// Mitsubishi GX Works2 project: BookEX6_22 Compare   PLC: Q13UDV

// global labels: Global
VAR_GLOBAL
  bVar0 AT M5000 : BOOL;
  abArray0 AT M5010 : ARRAY [0..49] OF BOOL;
  sStr0 AT D5000 : STRING[199];
  sStr1 AT D5100 : STRING[199];
  sStr2 AT D5200 : STRING[199];
  sStr3 AT D5300 : STRING[199];
  sStr4 AT D5400 : STRING[199];
  sStr5 AT D5500 : STRING[199];
  sStr6 AT D5600 : STRING[199];
  sStr7 AT D5700 : STRING[199];
  sStr8 AT D5800 : STRING[199];
  sStr9 AT D5900 : STRING[199];
  iVar0 AT D4500 : INT;
  iVar1 AT D4501 : INT;
  iVar2 AT D4502 : INT;
  iVar3 AT D4503 : INT;
  iVar4 AT D4504 : INT;
  iVar5 AT D4505 : INT;
  iVar6 AT D4506 : INT;
  iVar7 AT D4507 : INT;
  iVar8 AT D4508 : INT;
  iVar9 AT D4509 : INT;
  dVar0 AT D4510 : DINT;
  dVar1 AT D4512 : DINT;
  dVar2 AT D4514 : DINT;
  dVar3 AT D4516 : DINT;
  dVar4 AT D4518 : DINT;
  dVar5 AT D4520 : DINT;
  dVar6 AT D4522 : DINT;
  dVar7 AT D4524 : DINT;
  dVar8 AT D4526 : DINT;
  dVar9 AT D4528 : DINT;
  wVar0 AT D4530 : WORD;
  wVar1 AT D4531 : WORD;
  wVar2 AT D4532 : WORD;
  wVar3 AT D4533 : WORD;
  wVar4 AT D4534 : WORD;
  wVar5 AT D4535 : WORD;
  wVar6 AT D4536 : WORD;
  wVar7 AT D4537 : WORD;
  wVar8 AT D4538 : WORD;
  wVar9 AT D4539 : WORD;
  dwVar0 AT D4540 : DWORD;
  dwVar1 AT D4542 : DWORD;
  dwVar2 AT D4544 : DWORD;
  dwVar3 AT D4546 : DWORD;
  dwVar4 AT D4548 : DWORD;
  dwVar5 AT D4550 : DWORD;
  dwVar6 AT D4552 : DWORD;
  dwVar7 AT D4554 : DWORD;
  dwVar8 AT D4556 : DWORD;
  dwVar9 AT D4558 : DWORD;
  fsVar0 AT D4560 : REAL;
  fsVar1 AT D4562 : REAL;
  fsVar2 AT D4564 : REAL;
  fsVar3 AT D4566 : REAL;
  fsVar4 AT D4568 : REAL;
  fsVar5 AT D4570 : REAL;
  fsVar6 AT D4572 : REAL;
  fsVar7 AT D4574 : REAL;
  fsVar8 AT D4576 : REAL;
  fsVar9 AT D4578 : REAL;
  fdVar0 AT D4580 : LREAL;
  tTime0 AT D4620 : TIME;
  tTime1 AT D4622 : TIME;
  tTime2 AT D4624 : TIME;
  tTime3 AT D4626 : TIME;
  tTime4 AT D4628 : TIME;
  tTime5 AT D4630 : TIME;
  tTime6 AT D4632 : TIME;
  tTime7 AT D4634 : TIME;
  tTime8 AT D4636 : TIME;
  tTime9 AT D4638 : TIME;
  tTime10 AT D4640 : TIME;
  bVar1 AT M5001 : BOOL;
  bVar2 AT M5002 : BOOL;
  bVar3 AT M5003 : BOOL;
  bVar4 AT M5004 : BOOL;
  bVar5 AT M5005 : BOOL;
  bVar6 AT M5006 : BOOL;
  bVar7 AT M5007 : BOOL;
  bVar8 AT M5008 : BOOL;
  bVar9 AT M5009 : BOOL;
  abArray1 AT M5060 : ARRAY [0..49] OF BOOL;
  abArray2 AT M5110 : ARRAY [0..49] OF BOOL;
  abArray3 AT M5160 : ARRAY [0..49] OF BOOL;
  abArray4 AT M5210 : ARRAY [0..49] OF BOOL;
  abArray5 AT M5260 : ARRAY [0..49] OF BOOL;
  abArray6 AT M5310 : ARRAY [0..49] OF BOOL;
  abArray7 AT M5360 : ARRAY [0..49] OF BOOL;
  abArray8 AT M5410 : ARRAY [0..49] OF BOOL;
  abArray9 AT M5460 : ARRAY [0..49] OF BOOL;
  fdVar1 AT D4584 : LREAL;
  fdVar2 AT D4588 : LREAL;
  fdVar3 AT D4592 : LREAL;
  fdVar4 AT D4596 : LREAL;
  fdVar5 AT D4600 : LREAL;
  fdVar6 AT D4604 : LREAL;
  fdVar7 AT D4608 : LREAL;
  fdVar8 AT D4612 : LREAL;
  fdVar9 AT D4616 : LREAL;
  afsPen0 AT D2000 : ARRAY [0..499] OF REAL;
  afsPen1 AT D3000 : ARRAY [0..499] OF REAL;
END_VAR
// user libraries (not included): HMI

PROGRAM ExBKCMP
VAR
  Mov4WORD_1 : Mov4WORD;
  Mov4WORD_2 : Mov4WORD;
  Mov4WORD_0 : Mov4WORD;
  Mov4WORD_3 : Mov4WORD;
  Mov4WORD_4 : Mov4WORD;
END_VAR
(* structured ladder/FBD written out as ST: instructions are called as NAME(EN, inputs, outputs); _pN, _eN, _tN stand for wires *)
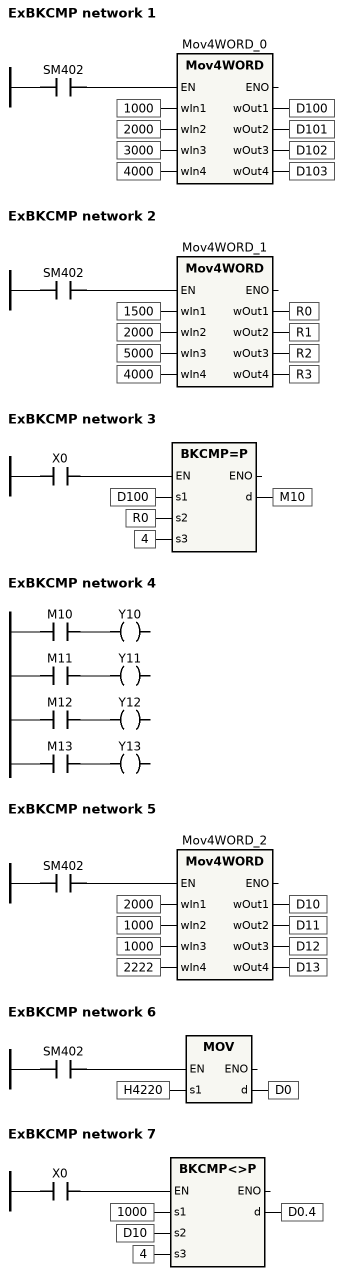
(* network 1 *)
Mov4WORD_0(EN := SM402, wIn1 := 1000, wIn2 := 2000, wIn3 := 3000, wIn4 := 4000, wOut1 => D100, wOut2 => D101, wOut3 => D102, wOut4 => D103);
(* network 2 *)
Mov4WORD_1(EN := SM402, wIn1 := 1500, wIn2 := 2000, wIn3 := 5000, wIn4 := 4000, wOut1 => R0, wOut2 => R1, wOut3 => R2, wOut4 => R3);
(* network 3 *)
BKCMP=P(X0, D100, R0, 4, M10);
(* network 4 *)
Y10 := M10;
Y11 := M11;
Y12 := M12;
Y13 := M13;
(* network 5 *)
Mov4WORD_2(EN := SM402, wIn1 := 2000, wIn2 := 1000, wIn3 := 1000, wIn4 := 2222, wOut1 => D10, wOut2 => D11, wOut3 => D12, wOut4 => D13);
(* network 6 *)
MOV(SM402, H4220, D0);
(* network 7 *)
BKCMP<>P(X0, 1000, D10, 4, D0.4);
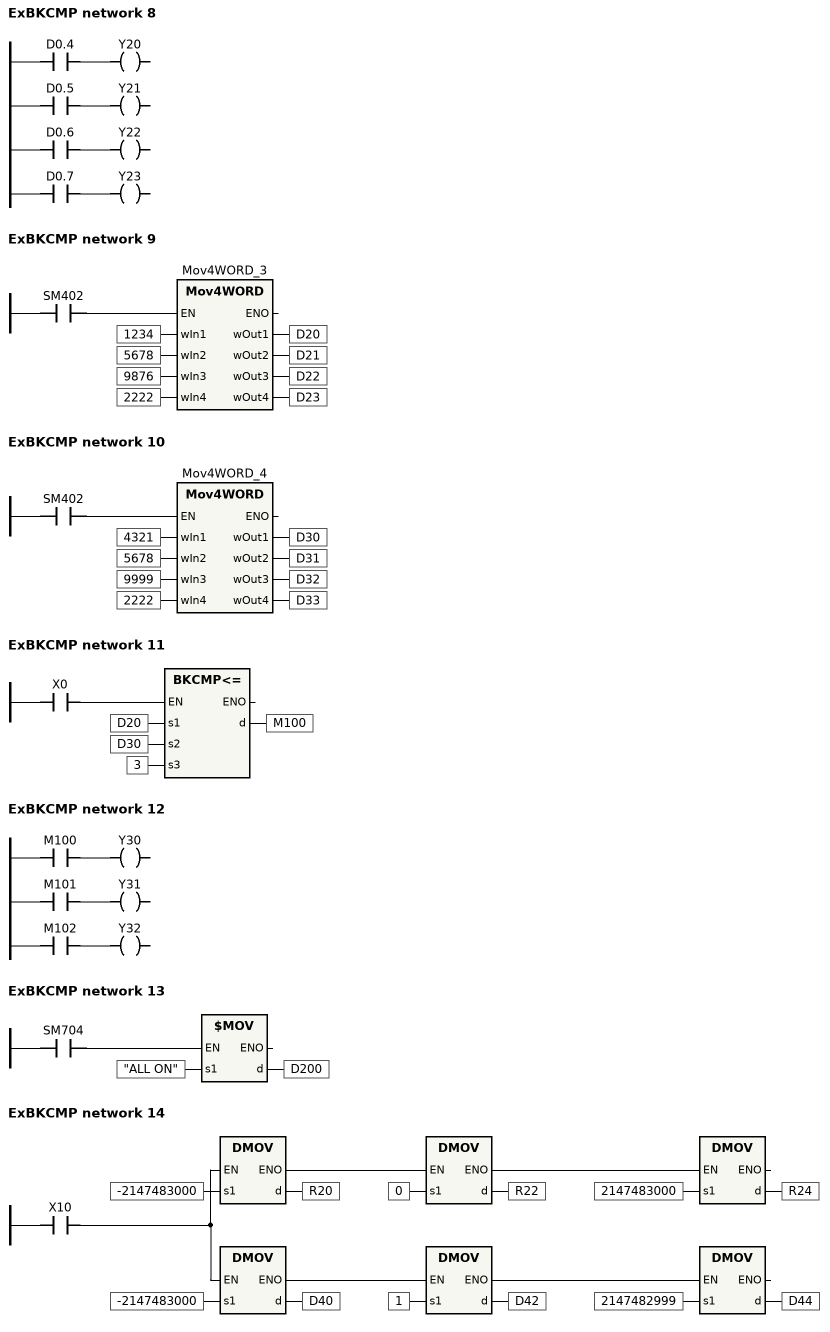
(* network 8 *)
Y20 := D0.4;
Y21 := D0.5;
Y22 := D0.6;
Y23 := D0.7;
(* network 9 *)
Mov4WORD_3(EN := SM402, wIn1 := 1234, wIn2 := 5678, wIn3 := 9876, wIn4 := 2222, wOut1 => D20, wOut2 => D21, wOut3 => D22, wOut4 => D23);
(* network 10 *)
Mov4WORD_4(EN := SM402, wIn1 := 4321, wIn2 := 5678, wIn3 := 9999, wIn4 := 2222, wOut1 => D30, wOut2 => D31, wOut3 => D32, wOut4 => D33);
(* network 11 *)
BKCMP<=(X0, D20, D30, 3, M100);
(* network 12 *)
Y30 := M100;
Y31 := M101;
Y32 := M102;
(* network 13 *)
$MOV(SM704, "ALL ON", D200);
(* network 14 *)
_e1 := DMOV(X10, -2147483000, R20);
_e2 := DMOV(_e1, 0, R22);
DMOV(_e2, 2147483000, R24);
_e3 := DMOV(X10, -2147483000, D40);
_e4 := DMOV(_e3, 1, D42);
DMOV(_e4, 2147482999, D44);
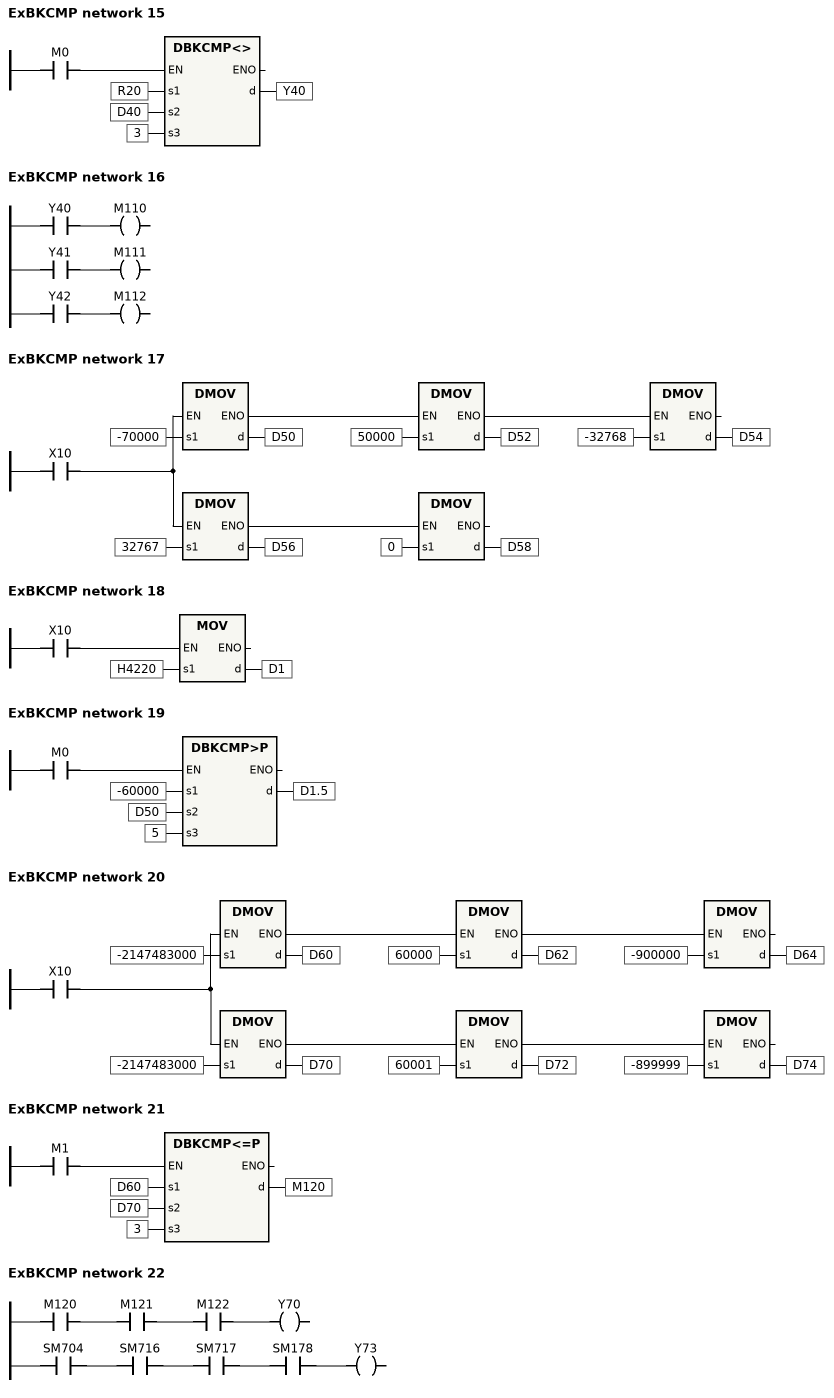
(* network 15 *)
DBKCMP<>(M0, R20, D40, 3, Y40);
(* network 16 *)
M110 := Y40;
M111 := Y41;
M112 := Y42;
(* network 17 *)
_e1 := DMOV(X10, -70000, D50);
_e2 := DMOV(_e1, 50000, D52);
DMOV(_e2, -32768, D54);
_e3 := DMOV(X10, 32767, D56);
DMOV(_e3, 0, D58);
(* network 18 *)
MOV(X10, H4220, D1);
(* network 19 *)
DBKCMP>P(M0, -60000, D50, 5, D1.5);
(* network 20 *)
_e1 := DMOV(X10, -2147483000, D60);
_e2 := DMOV(_e1, 60000, D62);
DMOV(_e2, -900000, D64);
_e3 := DMOV(X10, -2147483000, D70);
_e4 := DMOV(_e3, 60001, D72);
DMOV(_e4, -899999, D74);
(* network 21 *)
DBKCMP<=P(M1, D60, D70, 3, M120);
(* network 22 *)
Y70 := M120 AND M121 AND M122;
Y73 := SM704 AND SM716 AND SM717 AND SM178;
END_PROGRAM

PROGRAM ExCMP
VAR
  abRes : ARRAY [0..2] OF BOOL;
END_VAR
(* structured ladder/FBD written out as ST: instructions are called as NAME(EN, inputs, outputs); _pN, _eN, _tN stand for wires *)
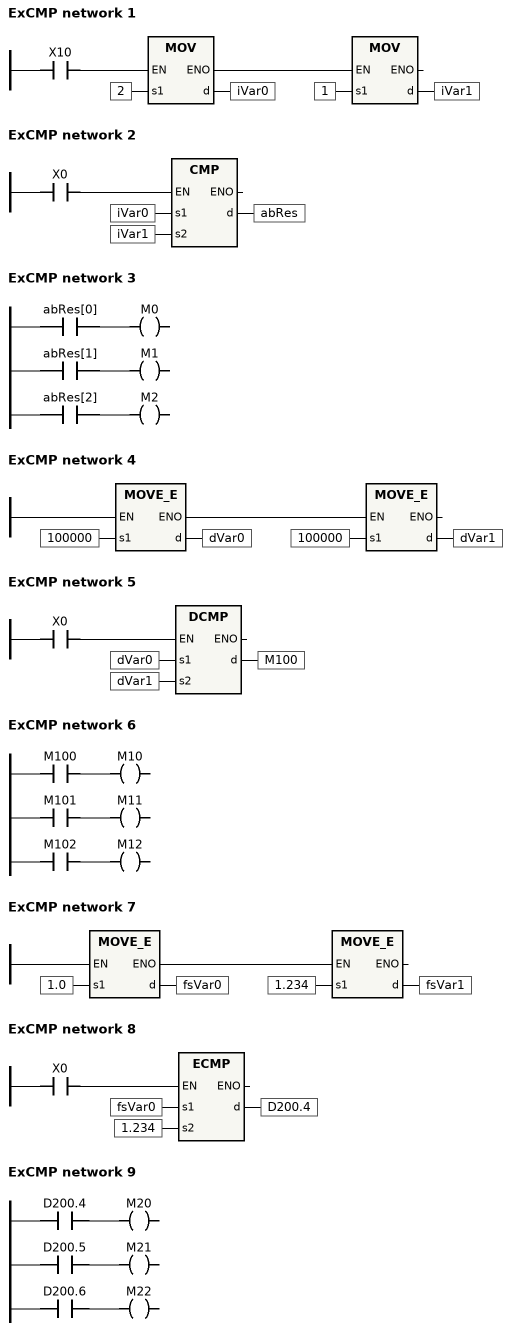
(* network 1 *)
_e1 := MOV(X10, 2, iVar0);
MOV(_e1, 1, iVar1);
(* network 2 *)
CMP(X0, iVar0, iVar1, abRes);
(* network 3 *)
M0 := abRes[0];
M1 := abRes[1];
M2 := abRes[2];
(* network 4 *)
_e1 := MOVE_E(TRUE, 100000, dVar0);
MOVE_E(_e1, 100000, dVar1);
(* network 5 *)
DCMP(X0, dVar0, dVar1, M100);
(* network 6 *)
M10 := M100;
M11 := M101;
M12 := M102;
(* network 7 *)
_e1 := MOVE_E(TRUE, 1.0, fsVar0);
MOVE_E(_e1, 1.234, fsVar1);
(* network 8 *)
ECMP(X0, fsVar0, 1.234, D200.4);
(* network 9 *)
M20 := D200.4;
M21 := D200.5;
M22 := D200.6;
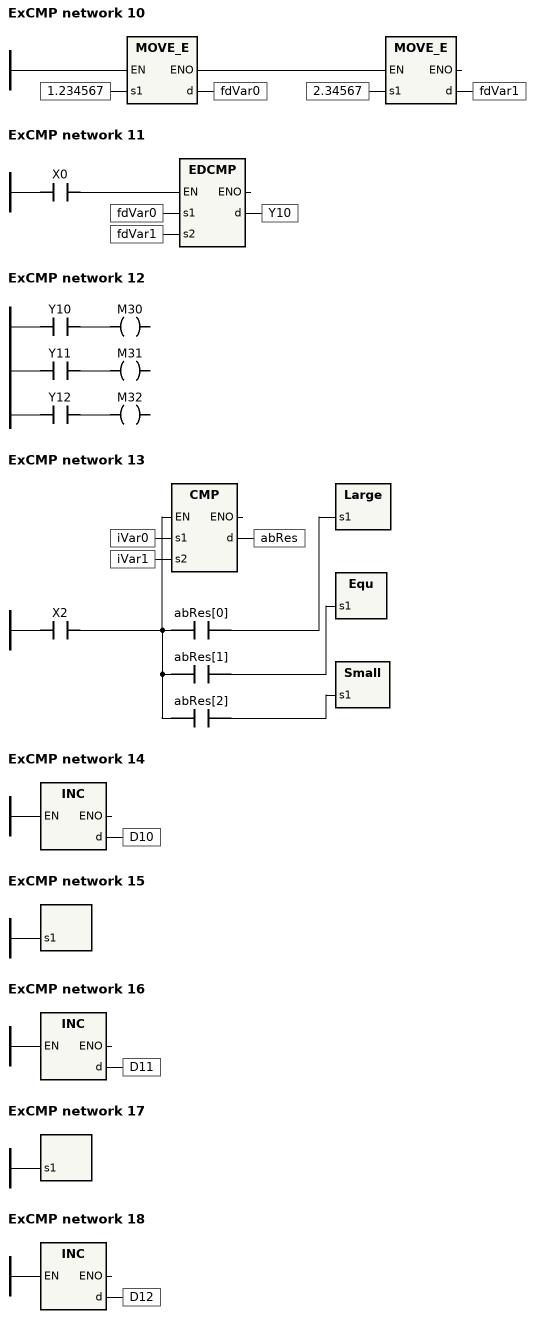
(* network 10 *)
_e1 := MOVE_E(TRUE, 1.234567, fdVar0);
MOVE_E(_e1, 2.34567, fdVar1);
(* network 11 *)
EDCMP(X0, fdVar0, fdVar1, Y10);
(* network 12 *)
M30 := Y10;
M31 := Y11;
M32 := Y12;
(* network 13 *)
CMP(X2, iVar0, iVar1, abRes);
(* element kind 9 Large <- X2 AND abRes[0] *)
(* element kind 9 Equ <- X2 AND abRes[1] *)
(* element kind 9 Small <- X2 AND abRes[2] *)
(* network 14 *)
INC(TRUE, D10);
(* network 15 *)
(* element kind 10  <- TRUE *)
(* network 16 Large: *)
INC(TRUE, D11);
(* network 17 *)
(* element kind 10  <- TRUE *)
(* network 18 Equ: *)
INC(TRUE, D12);
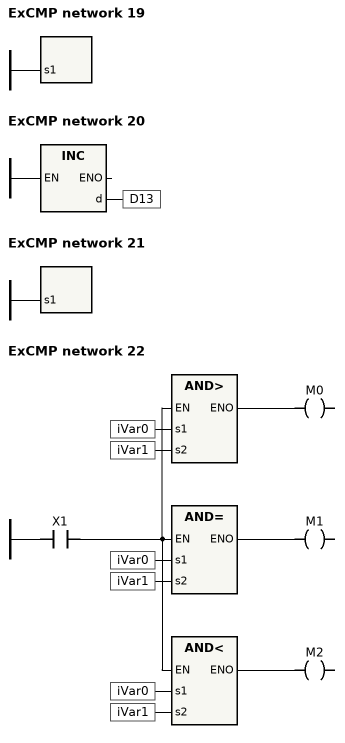
(* network 19 *)
(* element kind 10  <- TRUE *)
(* network 20 Small: *)
INC(TRUE, D13);
(* network 21 *)
(* element kind 10  <- TRUE *)
(* network 22 *)
_e1 := AND>(X1, iVar0, iVar1);
M0 := _e1;
_e2 := AND=(X1, iVar0, iVar1);
M1 := _e2;
_e3 := AND<(X1, iVar0, iVar1);
M2 := _e3;
END_PROGRAM

PROGRAM ExLD
(* structured ladder/FBD written out as ST: instructions are called as NAME(EN, inputs, outputs); _pN, _eN, _tN stand for wires *)
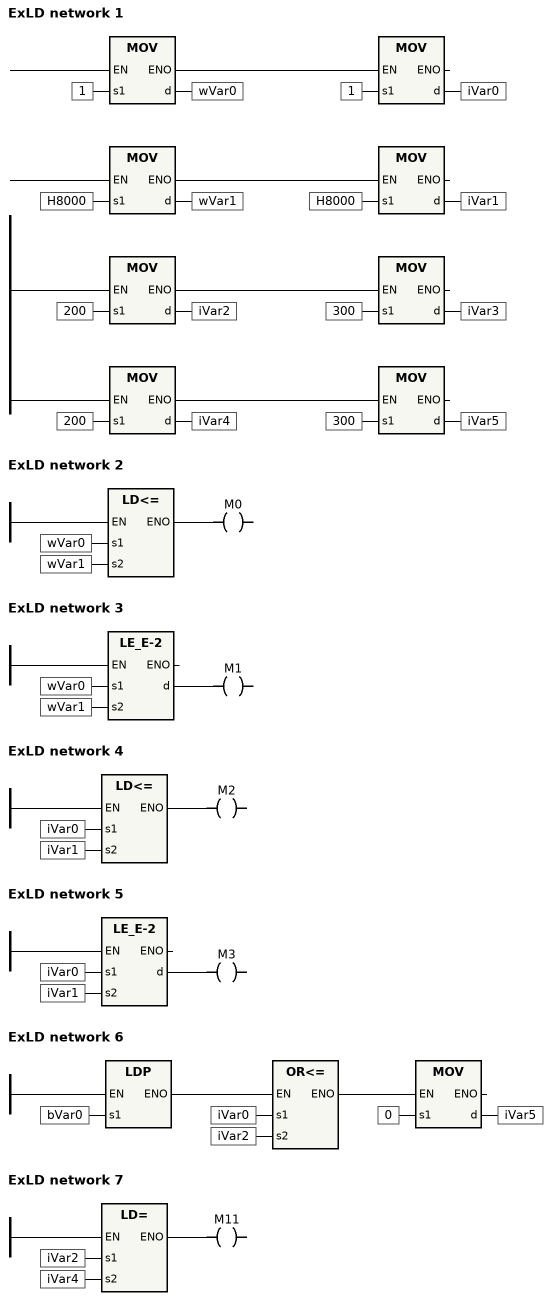
(* network 1 *)
_e1 := MOV(TRUE, 1, wVar0);
MOV(_e1, 1, iVar0);
_e2 := MOV(TRUE, H8000, wVar1);
MOV(_e2, H8000, iVar1);
_e3 := MOV(TRUE, 200, iVar2);
MOV(_e3, 300, iVar3);
_e4 := MOV(TRUE, 200, iVar4);
MOV(_e4, 300, iVar5);
(* network 2 *)
_e1 := LD<=(TRUE, wVar0, wVar1);
M0 := _e1;
(* network 3 *)
LE_E(TRUE, wVar0, wVar1, _t1);
M1 := _t1;
(* network 4 *)
_e1 := LD<=(TRUE, iVar0, iVar1);
M2 := _e1;
(* network 5 *)
LE_E(TRUE, iVar0, iVar1, _t1);
M3 := _t1;
(* network 6 *)
_e1 := LDP(TRUE, bVar0);
_e2 := OR<=(_e1, iVar0, iVar2);
MOV(_e2, 0, iVar5);
(* network 7 *)
_e1 := LD=(TRUE, iVar2, iVar4);
M11 := _e1;
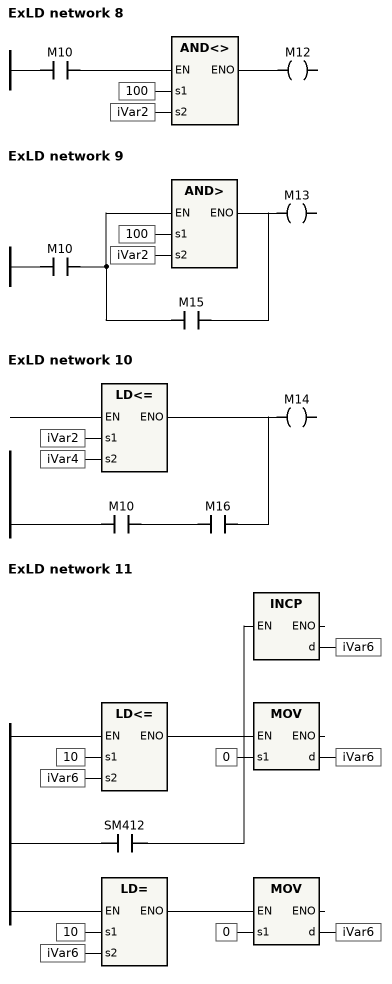
(* network 8 *)
_e1 := AND<>(M10, 100, iVar2);
M12 := _e1;
(* network 9 *)
_e1 := AND>(M10, 100, iVar2);
M13 := _e1 OR (M10 AND M15);
(* network 10 *)
_e1 := LD<=(TRUE, iVar2, iVar4);
M14 := (M10 AND M16) OR _e1;
(* network 11 *)
INCP(SM412, iVar6);
_e1 := LD<=(TRUE, 10, iVar6);
MOV(_e1, 0, iVar6);
_e2 := LD=(TRUE, 10, iVar6);
MOV(_e2, 0, iVar6);
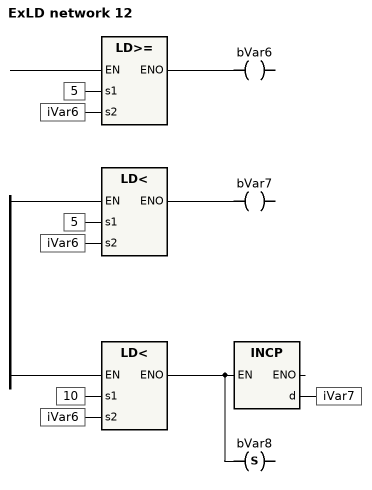
(* network 12 *)
_e1 := LD>=(TRUE, 5, iVar6);
bVar6 := _e1;
_e2 := LD<(TRUE, 5, iVar6);
bVar7 := _e2;
_e3 := LD<(TRUE, 10, iVar6);
SET(_e3, bVar8);
INCP(_e3, iVar7);
END_PROGRAM

PROGRAM ExLD$
(* structured ladder/FBD written out as ST: instructions are called as NAME(EN, inputs, outputs); _pN, _eN, _tN stand for wires *)
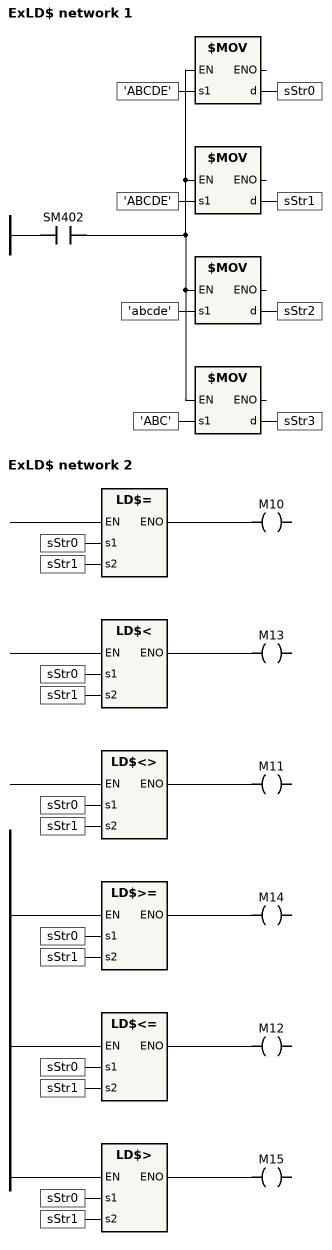
(* network 1 *)
$MOV(SM402, 'ABCDE', sStr0);
$MOV(SM402, 'ABCDE', sStr1);
$MOV(SM402, 'abcde', sStr2);
$MOV(SM402, 'ABC', sStr3);
(* network 2 *)
_e1 := LD$=(TRUE, sStr0, sStr1);
M10 := _e1;
_e2 := LD$<(TRUE, sStr0, sStr1);
M13 := _e2;
_e3 := LD$<>(TRUE, sStr0, sStr1);
M11 := _e3;
_e4 := LD$>=(TRUE, sStr0, sStr1);
M14 := _e4;
_e5 := LD$<=(TRUE, sStr0, sStr1);
M12 := _e5;
_e6 := LD$>(TRUE, sStr0, sStr1);
M15 := _e6;
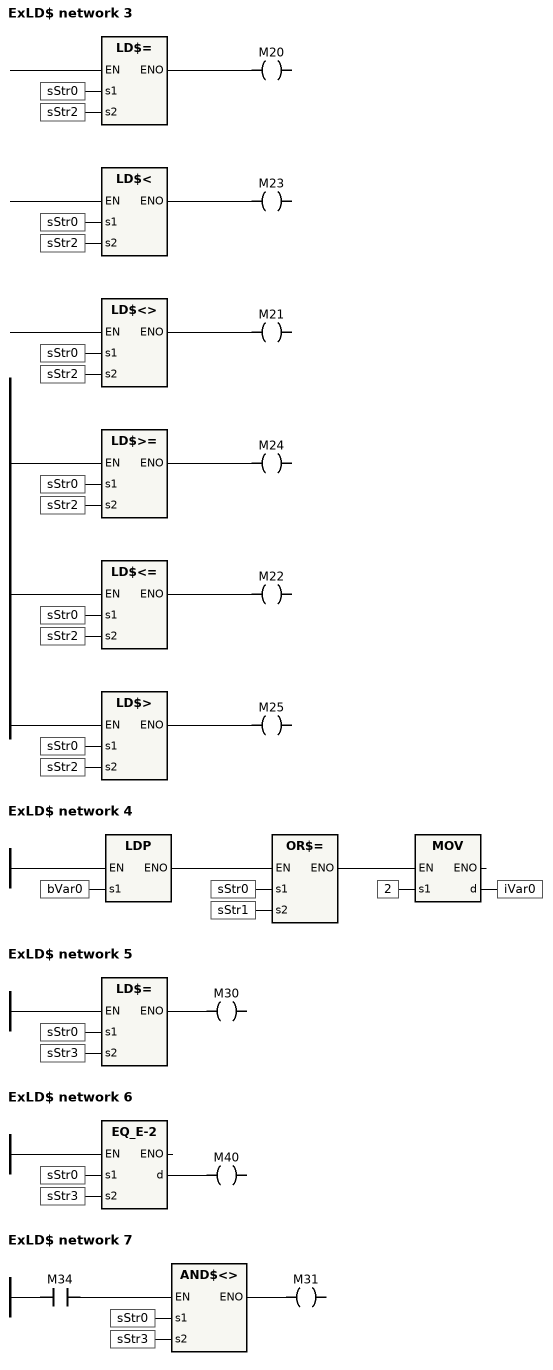
(* network 3 *)
_e1 := LD$=(TRUE, sStr0, sStr2);
M20 := _e1;
_e2 := LD$<(TRUE, sStr0, sStr2);
M23 := _e2;
_e3 := LD$<>(TRUE, sStr0, sStr2);
M21 := _e3;
_e4 := LD$>=(TRUE, sStr0, sStr2);
M24 := _e4;
_e5 := LD$<=(TRUE, sStr0, sStr2);
M22 := _e5;
_e6 := LD$>(TRUE, sStr0, sStr2);
M25 := _e6;
(* network 4 *)
_e1 := LDP(TRUE, bVar0);
_e2 := OR$=(_e1, sStr0, sStr1);
MOV(_e2, 2, iVar0);
(* network 5 *)
_e1 := LD$=(TRUE, sStr0, sStr3);
M30 := _e1;
(* network 6 *)
EQ_E(TRUE, sStr0, sStr3, _t1);
M40 := _t1;
(* network 7 *)
_e1 := AND$<>(M34, sStr0, sStr3);
M31 := _e1;
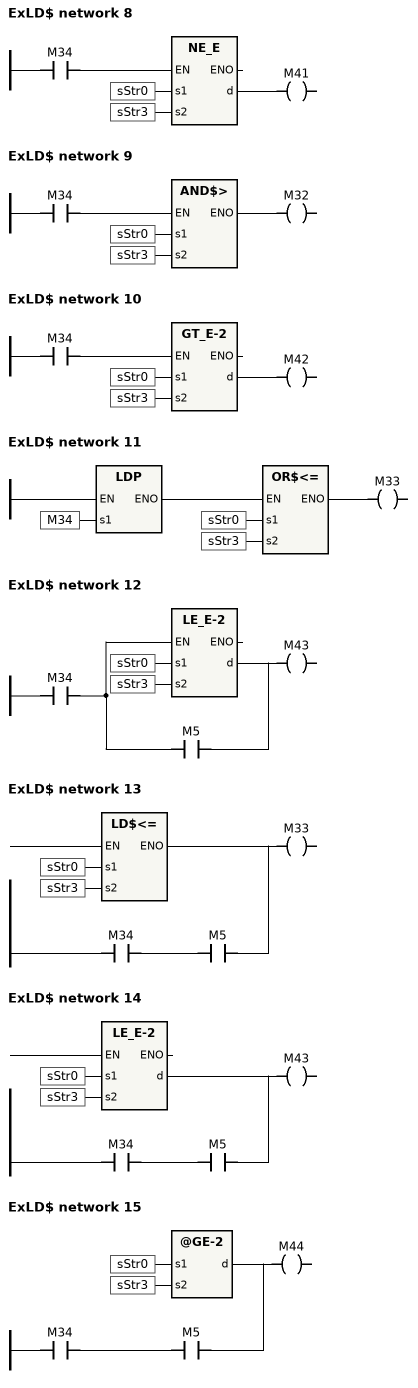
(* network 8 *)
NE_E(M34, sStr0, sStr3, _t1);
M41 := _t1;
(* network 9 *)
_e1 := AND$>(M34, sStr0, sStr3);
M32 := _e1;
(* network 10 *)
GT_E(M34, sStr0, sStr3, _t1);
M42 := _t1;
(* network 11 *)
_e1 := LDP(TRUE, M34);
_e2 := OR$<=(_e1, sStr0, sStr3);
M33 := _e2;
(* network 12 *)
LE_E(M34, sStr0, sStr3, _t1);
M43 := (M34 AND M5) OR _t1;
(* network 13 *)
_e1 := LD$<=(TRUE, sStr0, sStr3);
M33 := (M34 AND M5) OR _e1;
(* network 14 *)
LE_E(TRUE, sStr0, sStr3, _t1);
M43 := (M34 AND M5) OR _t1;
(* network 15 *)
M44 := (M34 AND M5) OR (@GE-2(sStr0, sStr3));
END_PROGRAM

PROGRAM ExLDD
(* structured ladder/FBD written out as ST: instructions are called as NAME(EN, inputs, outputs); _pN, _eN, _tN stand for wires *)
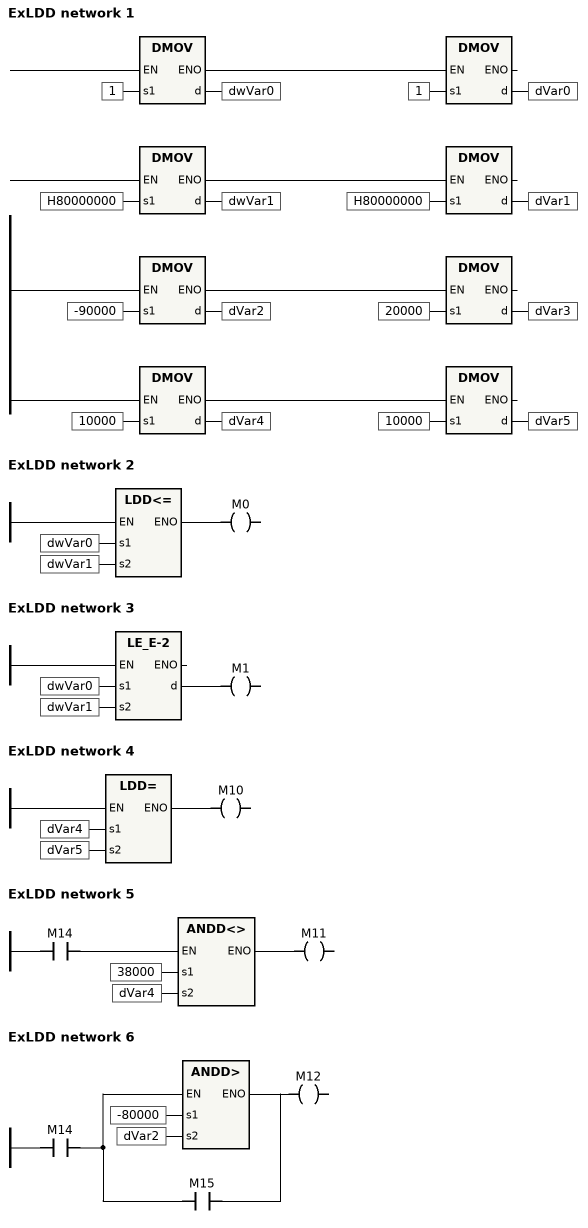
(* network 1 *)
_e1 := DMOV(TRUE, 1, dwVar0);
DMOV(_e1, 1, dVar0);
_e2 := DMOV(TRUE, H80000000, dwVar1);
DMOV(_e2, H80000000, dVar1);
_e3 := DMOV(TRUE, -90000, dVar2);
DMOV(_e3, 20000, dVar3);
_e4 := DMOV(TRUE, 10000, dVar4);
DMOV(_e4, 10000, dVar5);
(* network 2 *)
_e1 := LDD<=(TRUE, dwVar0, dwVar1);
M0 := _e1;
(* network 3 *)
LE_E(TRUE, dwVar0, dwVar1, _t1);
M1 := _t1;
(* network 4 *)
_e1 := LDD=(TRUE, dVar4, dVar5);
M10 := _e1;
(* network 5 *)
_e1 := ANDD<>(M14, 38000, dVar4);
M11 := _e1;
(* network 6 *)
_e1 := ANDD>(M14, -80000, dVar2);
M12 := _e1 OR (M14 AND M15);
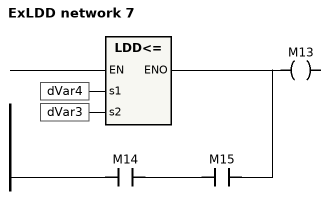
(* network 7 *)
_e1 := LDD<=(TRUE, dVar4, dVar3);
M13 := (M14 AND M15) OR _e1;
END_PROGRAM

PROGRAM ExLDE
(* structured ladder/FBD written out as ST: instructions are called as NAME(EN, inputs, outputs); _pN, _eN, _tN stand for wires *)
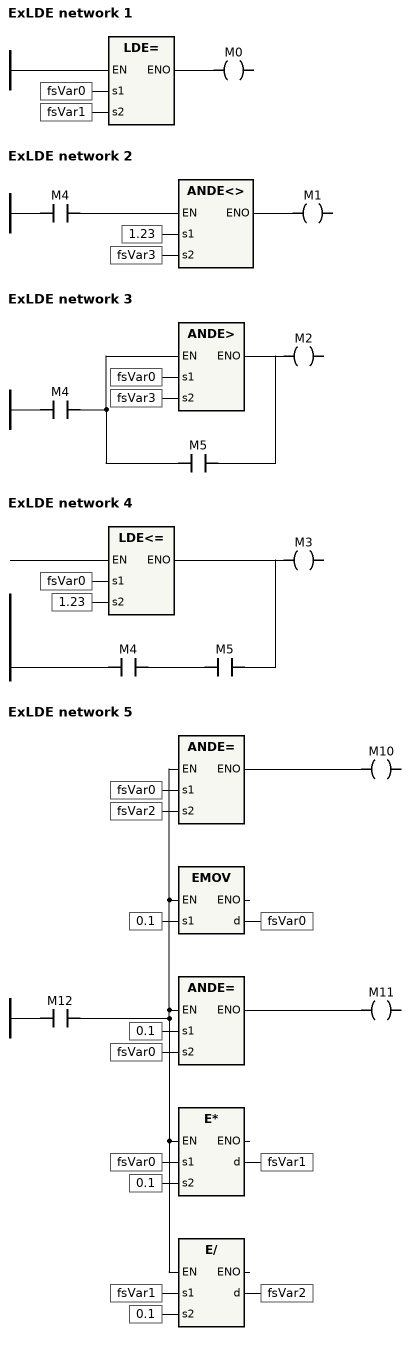
(* network 1 *)
_e1 := LDE=(TRUE, fsVar0, fsVar1);
M0 := _e1;
(* network 2 *)
_e1 := ANDE<>(M4, 1.23, fsVar3);
M1 := _e1;
(* network 3 *)
_e1 := ANDE>(M4, fsVar0, fsVar3);
M2 := _e1 OR (M4 AND M5);
(* network 4 *)
_e1 := LDE<=(TRUE, fsVar0, 1.23);
M3 := (M4 AND M5) OR _e1;
(* network 5 *)
EMOV(M12, 0.1, fsVar0);
E*(M12, fsVar0, 0.1, fsVar1);
E/(M12, fsVar1, 0.1, fsVar2);
_e1 := ANDE=(M12, fsVar0, fsVar2);
M10 := _e1;
_e2 := ANDE=(M12, 0.1, fsVar0);
M11 := _e2;
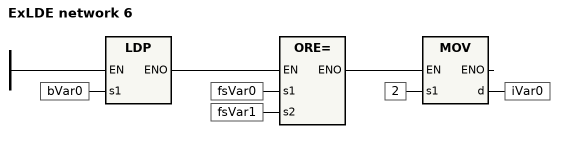
(* network 6 *)
_e1 := LDP(TRUE, bVar0);
_e2 := ORE=(_e1, fsVar0, fsVar1);
MOV(_e2, 2, iVar0);
END_PROGRAM

PROGRAM ExLDED
(* structured ladder/FBD written out as ST: instructions are called as NAME(EN, inputs, outputs); _pN, _eN, _tN stand for wires *)
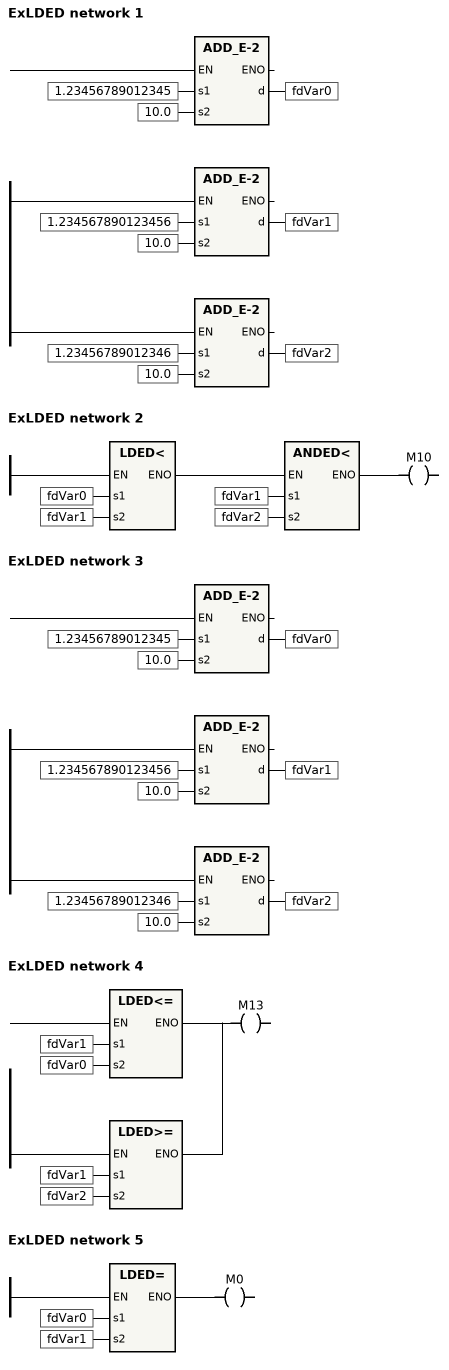
(* network 1 *)
ADD_E(TRUE, 1.23456789012345, 10.0, fdVar0);
ADD_E(TRUE, 1.234567890123456, 10.0, fdVar1);
ADD_E(TRUE, 1.23456789012346, 10.0, fdVar2);
(* network 2 *)
_e1 := LDED<(TRUE, fdVar0, fdVar1);
_e2 := ANDED<(_e1, fdVar1, fdVar2);
M10 := _e2;
(* network 3 *)
ADD_E(TRUE, 1.23456789012345, 10.0, fdVar0);
ADD_E(TRUE, 1.234567890123456, 10.0, fdVar1);
ADD_E(TRUE, 1.23456789012346, 10.0, fdVar2);
(* network 4 *)
_e1 := LDED<=(TRUE, fdVar1, fdVar0);
_e2 := LDED>=(TRUE, fdVar1, fdVar2);
M13 := _e1 OR _e2;
(* network 5 *)
_e1 := LDED=(TRUE, fdVar0, fdVar1);
M0 := _e1;
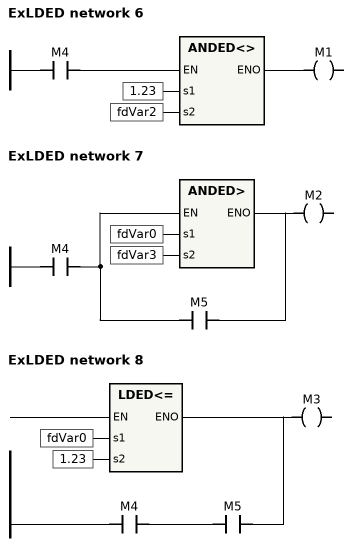
(* network 6 *)
_e1 := ANDED<>(M4, 1.23, fdVar2);
M1 := _e1;
(* network 7 *)
_e1 := ANDED>(M4, fdVar0, fdVar3);
M2 := _e1 OR (M4 AND M5);
(* network 8 *)
_e1 := LDED<=(TRUE, fdVar0, 1.23);
M3 := (M4 AND M5) OR _e1;
END_PROGRAM

PROGRAM ExZCP
VAR
  abRes : ARRAY [0..2] OF BOOL;
END_VAR
(* structured ladder/FBD written out as ST: instructions are called as NAME(EN, inputs, outputs); _pN, _eN, _tN stand for wires *)
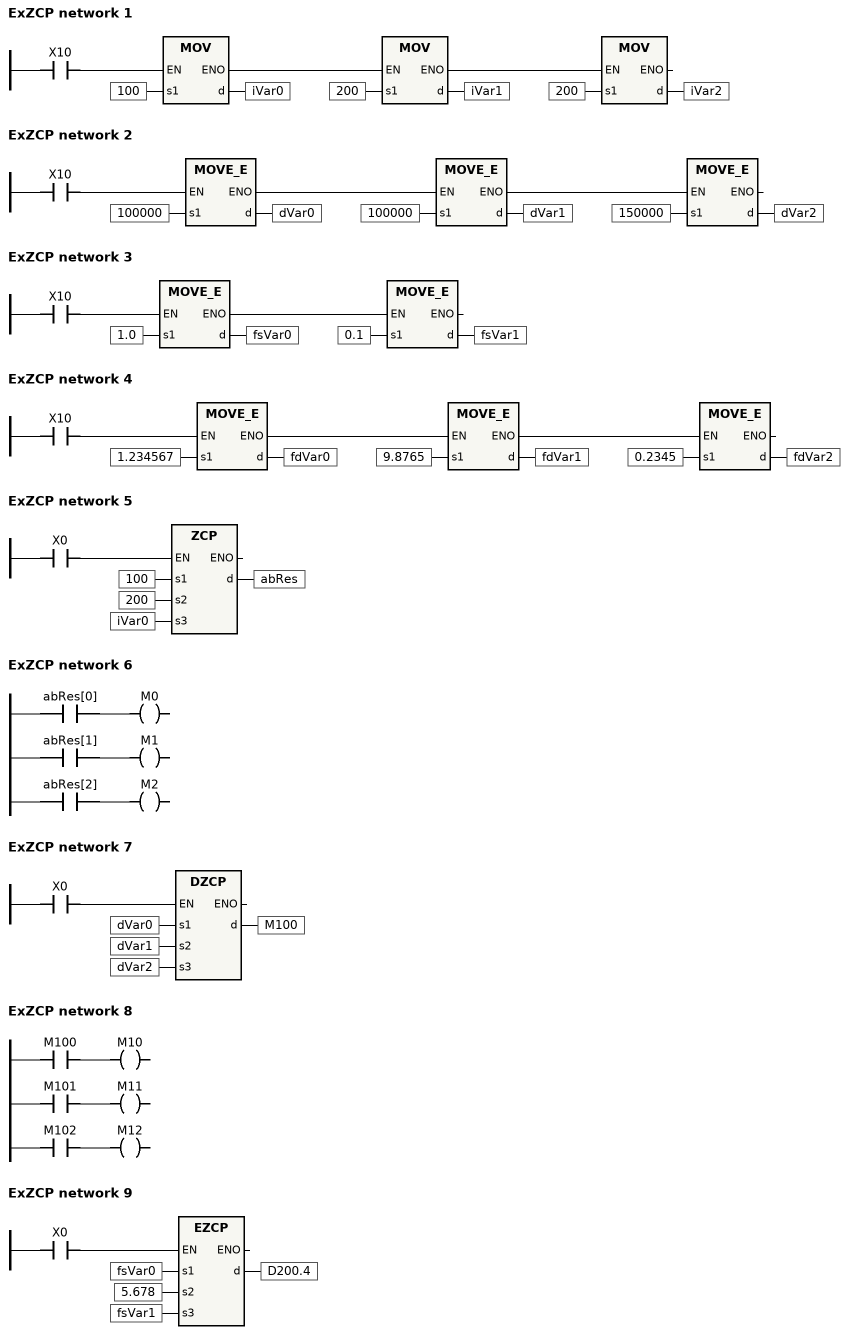
(* network 1 *)
_e1 := MOV(X10, 100, iVar0);
_e2 := MOV(_e1, 200, iVar1);
MOV(_e2, 200, iVar2);
(* network 2 *)
_e1 := MOVE_E(X10, 100000, dVar0);
_e2 := MOVE_E(_e1, 100000, dVar1);
MOVE_E(_e2, 150000, dVar2);
(* network 3 *)
_e1 := MOVE_E(X10, 1.0, fsVar0);
MOVE_E(_e1, 0.1, fsVar1);
(* network 4 *)
_e1 := MOVE_E(X10, 1.234567, fdVar0);
_e2 := MOVE_E(_e1, 9.8765, fdVar1);
MOVE_E(_e2, 0.2345, fdVar2);
(* network 5 *)
ZCP(X0, 100, 200, iVar0, abRes);
(* network 6 *)
M0 := abRes[0];
M1 := abRes[1];
M2 := abRes[2];
(* network 7 *)
DZCP(X0, dVar0, dVar1, dVar2, M100);
(* network 8 *)
M10 := M100;
M11 := M101;
M12 := M102;
(* network 9 *)
EZCP(X0, fsVar0, 5.678, fsVar1, D200.4);
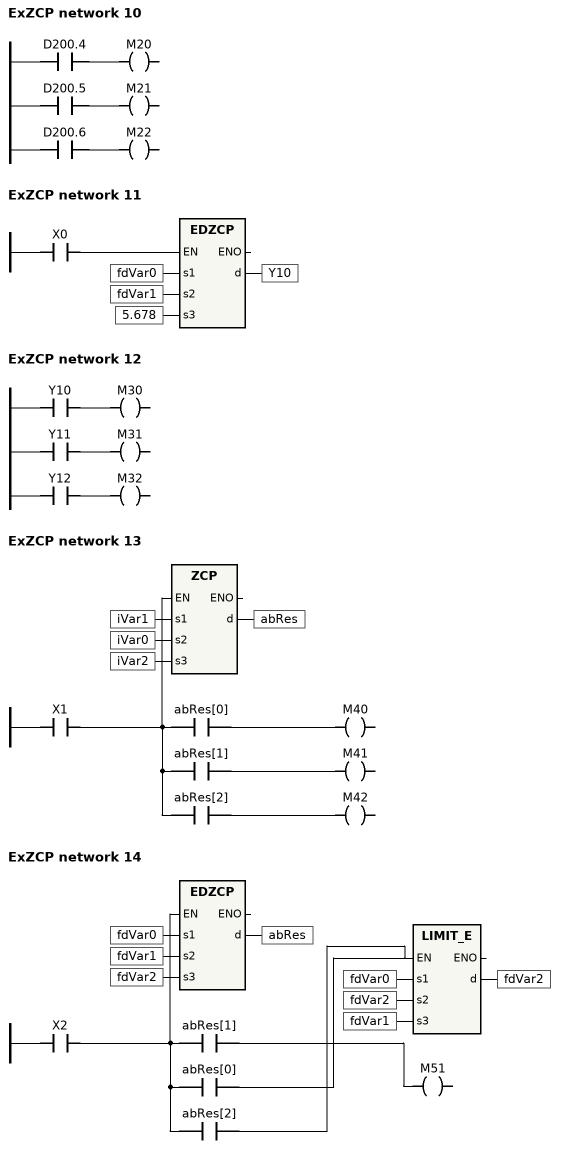
(* network 10 *)
M20 := D200.4;
M21 := D200.5;
M22 := D200.6;
(* network 11 *)
EDZCP(X0, fdVar0, fdVar1, 5.678, Y10);
(* network 12 *)
M30 := Y10;
M31 := Y11;
M32 := Y12;
(* network 13 *)
ZCP(X1, iVar1, iVar0, iVar2, abRes);
M40 := X1 AND abRes[0];
M41 := X1 AND abRes[1];
M42 := X1 AND abRes[2];
(* network 14 *)
EDZCP(X2, fdVar0, fdVar1, fdVar2, abRes);
M51 := X2 AND abRes[1];
LIMIT_E((X2 AND abRes[0]) OR (X2 AND abRes[2]), fdVar0, fdVar2, fdVar1, fdVar2);
END_PROGRAM
